PROGRAM RobotDynamics

VAR
	// slave robot arms joint data
	m_slaveJointsData AT %I* :ST_SlaveJointData;
	
	// setup joint5 position
	m_setupJointData AT %I* :ST_SetupJointData;
	
	// setup arms infromation;
	m_setupStatus AT %I* : ST_SetupStatus;
	
	// instrument info
	m_instruInfo AT %I* :ARRAY[1..g_sArmNum] OF ST_InstruStatus;
	
	// dynamic output
	m_slaveDynaData AT %Q* : ST_SlaveDynaData;
	m_setupJnt3Gravity AT %Q* : ARRAY[1..g_sArmNum] OF LREAL;
	m_setupJnt5Gravity AT %Q* : ARRAY[1..g_sArmNum] OF LREAL;
	
	// flag to init robot dynamic model
	m_robotDynaInit :BOOL :=FALSE;
	
	// grivity model block
	m_slaveGravityModel :ARRAY[1..g_sArmNum] OF FB_SlaveGravity;
	m_setupGravityModel :ARRAY[1..g_sArmNum] OF FB_SetupGravity;
	
	// slave dynamic block
	m_slaveDynamicModel :ARRAY[1..g_sArmNum] OF FB_SlaveDynamic;
	
	// instument out-of-view check
	m_instruViewCheck :FB_InstruViewCheck;
	
	// slave arm self-collision avoidance
	m_selfCollisonAvoid : FB_SelfCollisionAvoid;
	
	// code execute time measure
	m_codeTime : Profiler;
	
	// tmp variables
	i: INT;
	
END_VAR

m_codeTime(START:=TRUE, RESET:=TRUE);

// wait config file loaded
IF NOT(SafetyCheck.m_loadConfigFileOK) OR NOT(slaveArmControl.m_robotInit) OR NOT(SetupArmControl.m_robotInit) THEN
	RETURN;
END_IF

// robot dynamic model init
IF m_robotDynaInit =FALSE THEN
	FOR i:=1 TO g_sArmNum DO
		m_slaveGravityModel[i].Init(i);
		m_setupGravityModel[i].init(i);
		m_slaveDynamicModel[i].init(i);
	END_FOR
	m_instruViewCheck.init();
	m_selfCollisonAvoid.init();

	m_robotDynaInit:=TRUE;
END_IF


FOR i:=1 TO g_sArmNum DO
	// run gravity model
	m_slaveDynaData.m_gravity[i]:=m_slaveGravityModel[i].run(m_setupJointData.m_curJntPos[i][5], m_slaveJointsData.m_curJntPos[i],m_instruInfo[i]);
	m_setupGravityModel[i].run(m_setupJointData.m_curJntPos[i], m_slaveJointsData.m_curJntPos[i],m_instruInfo[i], o_jnt3Gravity=> m_setupJnt3Gravity[i], o_jnt5Gravity=> m_setupJnt5Gravity[i]);
	
	// run dynamic model
	m_slaveDynamicModel[i].updateDynamic(m_slaveJointsData.m_curJntPos[i]);
	m_slaveDynaData.m_massMat[i]:= m_slaveDynamicModel[i].jntMassMat;
END_FOR

m_instruViewCheck.run(m_setupJointData.m_curJntPos, m_slaveJointsData.m_curDHJntPos, m_instruInfo);
m_slaveDynaData.m_insruViewData:=m_instruViewCheck.m_instruImgBoundPos;

m_selfCollisonAvoid.run(m_setupStatus.m_curEndPose,m_slaveJointsData.m_curDHJntPos, o_repulseJntVel=>m_slaveDynaData.m_repulseJntVel);

m_codeTime(START:=FALSE);

END_PROGRAM

(* stored: Version 1.1.0.1, ProductVersion 3.1.4024.11
   POU RobotDynamics: Id {798b314f-0a53-4e08-997d-5fefed426c86}, SpecialFunc None *)
